Staubli VAL3: refresh.pgx

program refresh()
// // page refresh
  local string l_sMessage
begin
  // check the page
  if !bPage
    if !bShowMessage
      if (nKey>=270 and nKey<=278)or abs(clock()-nRefresh)>nTime or use:bUseRefresh
        if (nKey>=270 and nKey<=278)or use:bUseRefresh
          cls()
        endIf
        // refresh the static message
        use:bUseRefresh=true
        call refreshStatic()
        call refreshDynamic()
        // update the clock
        nRefresh=clock()
      else
        // refresh the Dynamic message
        call refreshDynamic()
      endIf
    endIf
    // print the message
    call showMessage()
  else
    call showLog()
  endIf
  call printToShow()
end
